// TIA Portal project "CarBeltLift" (V15.1)

(* hardware
DEVICE "S71500/ET200MP-Station_1"  S7-1500 station
   slot 0: "Profilschiene_0"  Rack  6ES7 590-1***0-0AA0
   slot 1: "PLC_1"  CPU 1513-1 PN  6ES7 513-1AL02-0AB0  V2.6
      slot 3: "CPU-Display_1"  6ES7591-1AA00-0AA0
   slot 2: "DI 16x24VDC BA_1"  DI 16x24VDC BA  6ES7 521-1BH10-0AA0  V1.0
   slot 3: "AI 4xU/I/RTD/TC ST_1"  AI 4xU/I/RTD/TC ST  6ES7 531-7QD00-0AB0  V1.0
   slot 4: "DQ 16x24VDC/0.5A BA_1"  DQ 16x24VDC/0.5A BA  6ES7 522-1BH10-0AA0  V1.0
   slot 5: "AQ 2xU/I ST_1"  AQ 2xU/I ST  6ES7 532-5NB00-0AB0  V1.0
   slot 6: "DI 16x24VDC BA_2"  DI 16x24VDC BA  6ES7 521-1BH10-0AA0  V1.0
*)

// ===== PLC "PLC_1"  CPU 1513-1 PN =====

VAR_GLOBAL   // PLC tag table "Standard-Variablentabelle"
   "ControlOn" AT %M0.0 : Bool;
   "Step1" AT %M0.1 : Bool;
   "Step2" AT %M0.2 : Bool;
   "Step3" AT %M0.3 : Bool;
   "Step4" AT %M0.4 : Bool;
   "StepsActive" AT %M0.5 : Bool;
   "GetLiftAbsTargetPosOk" AT %M0.6 : Bool;
   "StartAutoEdgeFlag" AT %M0.7 : Bool;
END_VAR

VAR_GLOBAL   // PLC tag table "Variablentabelle aus XML_1"
   "S1ControlOnPushButton" AT %I0.0 : Bool;
   "S2ControlOffPushButton" AT %I0.1 : Bool;   // NC
   "B1CarPosInLift" AT %I0.2 : Bool;   // NC
   "P1ControlOn" AT %Q0.0 : Bool;
   "M1Lift" AT %Q0.1 : Bool;
   "B2LiftPosMin" AT %I0.3 : Bool;   // NC
   "B4LiftPosAbs" AT %IW2 : Word;
   "B3LiftPosMax" AT %I0.4 : Bool;   // NC
   "LiftGoToNewPos" AT %Q0.4 : Bool;
   "LiftTargetPosAbs" AT %QW2 : Word;
   "LiftNewPosReached" AT %I0.5 : Bool;
   "M2ConvBeltToLift" AT %Q0.2 : Bool;
   "M3ConvBeltLift" AT %Q0.3 : Bool;
   "B5CarLevel1" AT %I0.6 : Bool;
   "B6CarLevel2" AT %I0.7 : Bool;
   "S3StartAuto" AT %I1.0 : Bool;
   "TargetLevel" AT %IW4 : Word;
END_VAR

FUNCTION "LiftSteps" : Void   // FC1, FBD
{ S7_Optimized_Access := 'TRUE' }
VERSION : 0.1
   VAR_TEMP   // added for the SCL form of the ladder/FBD networks
      _w1 : Bool;
   END_VAR
BEGIN

REGION Network 1: Start: M2 and M3 on
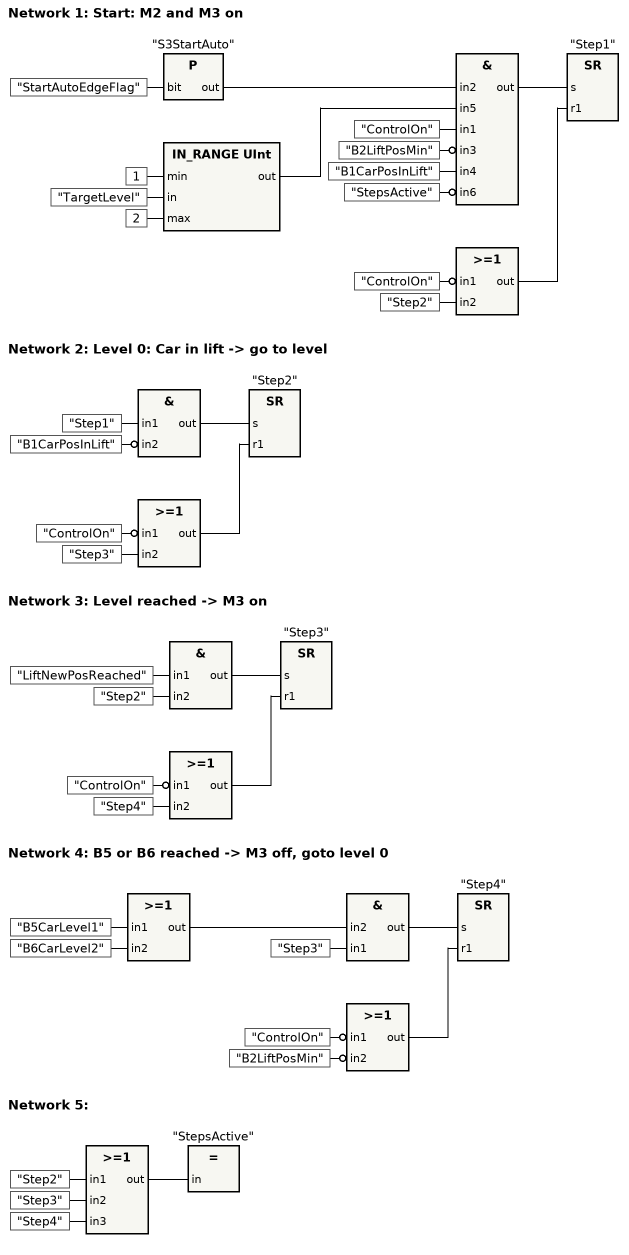
   #_w1 := "S3StartAuto" AND NOT "StartAutoEdgeFlag";   // rising edge of "S3StartAuto"
   "StartAutoEdgeFlag" := "S3StartAuto";
   IF #_w1 AND (1 <= "TargetLevel") AND ("TargetLevel" <= 2) AND "ControlOn" AND NOT "B2LiftPosMin" AND "B1CarPosInLift" AND NOT "StepsActive" THEN
       "Step1" := TRUE;   // SR flip-flop
   END_IF;
   IF NOT "ControlOn" OR "Step2" THEN "Step1" := FALSE; END_IF;
END_REGION

REGION Network 2: Level 0: Car in lift -> go to level
   IF "Step1" AND NOT "B1CarPosInLift" THEN
       "Step2" := TRUE;   // SR flip-flop
   END_IF;
   IF NOT "ControlOn" OR "Step3" THEN "Step2" := FALSE; END_IF;
END_REGION

REGION Network 3: Level reached -> M3 on
   IF "LiftNewPosReached" AND "Step2" THEN
       "Step3" := TRUE;   // SR flip-flop
   END_IF;
   IF NOT "ControlOn" OR "Step4" THEN "Step3" := FALSE; END_IF;
END_REGION

REGION Network 4: B5 or B6 reached -> M3 off, goto level 0
   IF ("B5CarLevel1" OR "B6CarLevel2") AND "Step3" THEN
       "Step4" := TRUE;   // SR flip-flop
   END_IF;
   IF NOT "ControlOn" OR NOT "B2LiftPosMin" THEN "Step4" := FALSE; END_IF;
END_REGION

REGION Network 5
   "StepsActive" := "Step2" OR "Step3" OR "Step4";
END_REGION
END_FUNCTION

FUNCTION "LiftSettings" : Void   // FC2, FBD
{ S7_Optimized_Access := 'TRUE' }
VERSION : 0.1
   VAR_TEMP   // added for the SCL form of the ladder/FBD networks
      _w1 : Bool;
   END_VAR
BEGIN

REGION Network 1
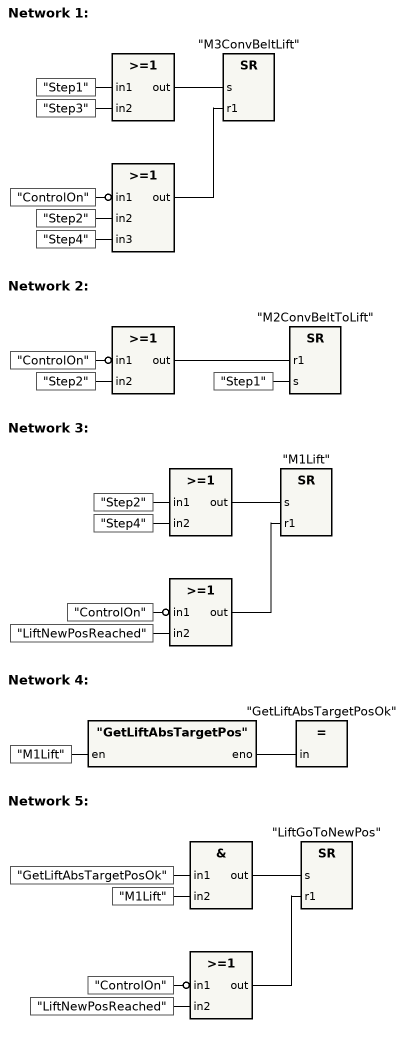
   IF "Step1" OR "Step3" THEN
       "M3ConvBeltLift" := TRUE;   // SR flip-flop
   END_IF;
   IF NOT "ControlOn" OR "Step2" OR "Step4" THEN "M3ConvBeltLift" := FALSE; END_IF;
END_REGION

REGION Network 2
   IF "Step1" THEN
       "M2ConvBeltToLift" := TRUE;   // SR flip-flop
   END_IF;
   IF NOT "ControlOn" OR "Step2" THEN "M2ConvBeltToLift" := FALSE; END_IF;
END_REGION

REGION Network 3
   IF "Step2" OR "Step4" THEN
       "M1Lift" := TRUE;   // SR flip-flop
   END_IF;
   IF NOT "ControlOn" OR "LiftNewPosReached" THEN "M1Lift" := FALSE; END_IF;
END_REGION

REGION Network 4
   "GetLiftAbsTargetPos"(EN := "M1Lift", ENO => #_w1);
   "GetLiftAbsTargetPosOk" := #_w1;
END_REGION

REGION Network 5
   IF "GetLiftAbsTargetPosOk" AND "M1Lift" THEN
       "LiftGoToNewPos" := TRUE;   // SR flip-flop
   END_IF;
   IF NOT "ControlOn" OR "LiftNewPosReached" THEN "LiftGoToNewPos" := FALSE; END_IF;
END_REGION
END_FUNCTION

FUNCTION "GetLiftAbsTargetPos" : Void   // FC3, FBD
{ S7_Optimized_Access := 'TRUE' }
VERSION : 0.1
   VAR_TEMP
      TargetLevelIntern : UInt;
   END_VAR
BEGIN

REGION Network 1
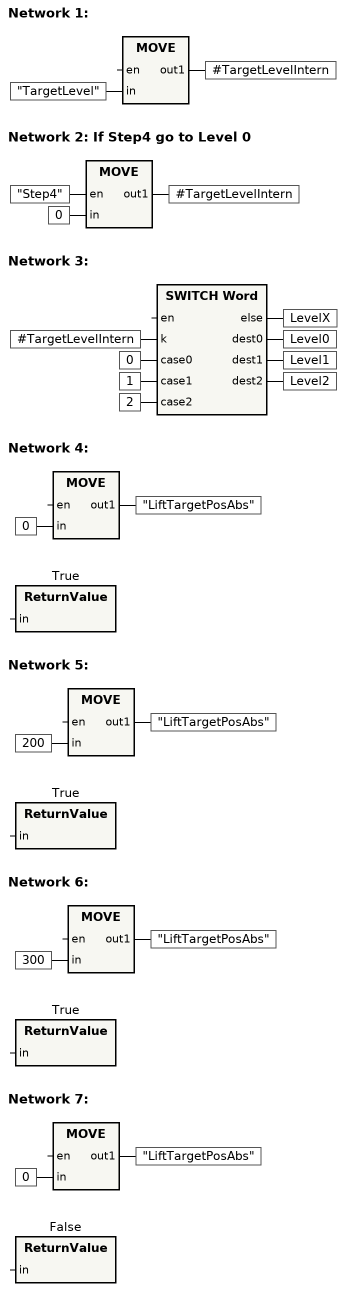
   #TargetLevelIntern := "TargetLevel";
END_REGION

REGION Network 2: If Step4 go to Level 0
   IF "Step4" THEN #TargetLevelIntern := 0; END_IF;
END_REGION

REGION Network 3
   // no SCL statement known for Switch: written as a call
   Switch(k := #TargetLevelIntern,
          case0 := 0,
          case1 := 1,
          case2 := 2,
          "else" => LevelX,
          dest0 => Level0,
          dest1 => Level1,
          dest2 => Level2);
END_REGION

REGION Network 4
   Level0:
   "LiftTargetPosAbs" := 0;
   ENO := True;
   RETURN;
END_REGION

REGION Network 5
   Level1:
   "LiftTargetPosAbs" := 200;
   ENO := True;
   RETURN;
END_REGION

REGION Network 6
   Level2:
   "LiftTargetPosAbs" := 300;
   ENO := True;
   RETURN;
END_REGION

REGION Network 7
   LevelX:
   "LiftTargetPosAbs" := 0;
   ENO := False;
   RETURN;
END_REGION
END_FUNCTION

FUNCTION "MHJ-PLC-Lab-Function-S71500" : Void   // FC4, SCL
{ S7_Optimized_Access := 'TRUE' }
VERSION : 0.1
   VAR_INPUT
      MinDiByte : Int;
      MaxDiByte : Int;
   END_VAR
   VAR_TEMP
      Value : Byte;
      ForCounter : Int;
      MaxDiByteTemp : Int;
      MinDiByteTemp : Int;
   END_VAR
   VAR CONSTANT
      Value_01_DW : DWord := 16#1223_5486;
      Value_02_DW : DWord := 16#A6C9_D1F5;
   END_VAR
BEGIN

   #Value:=PEEK(area := 16#82,
        dbNumber := 0,
        byteOffset := 511);
   #Value := #Value + 1;

   POKE(area := 16#82,
        dbNumber := 0,
        byteOffset := 511,
        value := #Value);

   POKE(area := 16#82,
        dbNumber := 0,
        byteOffset := 1016,
        value := #Value_01_DW);
   POKE(area := 16#82,
        dbNumber := 0,
        byteOffset := 1020,
        value := #Value_02_DW);

   #MaxDiByteTemp := 462;
   IF #MaxDiByte < 463 THEN
       #MaxDiByteTemp := #MaxDiByte;
   END_IF;

   #MinDiByteTemp := 0;
   IF #MaxDiByteTemp >= #MinDiByte & #MinDiByte >= 0 THEN
       #MinDiByteTemp := #MinDiByte;
   END_IF;

   FOR #ForCounter := #MinDiByteTemp TO #MaxDiByteTemp DO
       #Value := PEEK(area := 16#1,
                      dbNumber := 0,
                      byteOffset := #ForCounter);
       POKE(area := 16#81,
            dbNumber := 0,
            byteOffset := #ForCounter,
            value := #Value);
   END_FOR;

   #Value := PEEK(area := 16#1,
                  dbNumber := 0,
                  byteOffset := 512);
   POKE(area := 16#82,
        dbNumber := 0,
        byteOffset := 512,
        value := #Value);
END_FUNCTION

ORGANIZATION_BLOCK "Main"   // OB1, FBD, ProgramCycle
TITLE = "Main Program Sweep (Cycle)"
{ S7_Optimized_Access := 'TRUE' }
VERSION : 0.1
   VAR_INPUT
      Initial_Call : Bool;   // Initial call of this OB
      Remanence : Bool;   // =True, if remanent data are available
   END_VAR
BEGIN

REGION Network 1
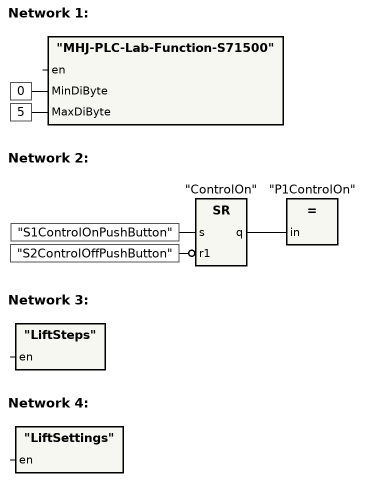
   "MHJ-PLC-Lab-Function-S71500"(MinDiByte := 0, MaxDiByte := 5);
END_REGION

REGION Network 2
   IF "S1ControlOnPushButton" THEN
       "ControlOn" := TRUE;   // SR flip-flop
   END_IF;
   IF NOT "S2ControlOffPushButton" THEN "ControlOn" := FALSE; END_IF;
   "P1ControlOn" := "ControlOn";
END_REGION

REGION Network 3
   "LiftSteps"();
END_REGION

REGION Network 4
   "LiftSettings"();
END_REGION
END_ORGANIZATION_BLOCK